FUNCTION_BLOCK EventWrapper_JACK2 (* Composite Function Block Type *)
  (* Standard: 61499-2 *)
  (* Version 0.0, 4/9/2019, erik, nxtControl GmbH, template *)
  PACKAGE Main;
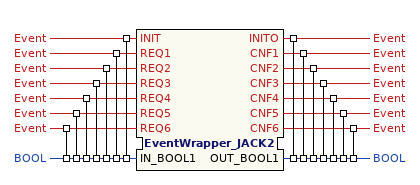
  EVENT_INPUT
    INIT WITH IN_BOOL1; (* Initialization Request *)
    REQ1 WITH IN_BOOL1; (* Normal Execution Request *)
    REQ2 WITH IN_BOOL1;
    REQ3 WITH IN_BOOL1;
    REQ4 WITH IN_BOOL1;
    REQ5 WITH IN_BOOL1;
    REQ6 WITH IN_BOOL1;
  END_EVENT
  EVENT_OUTPUT
    INITO WITH OUT_BOOL1; (* Initialization Confirm *)
    CNF1 WITH OUT_BOOL1; (* Execution Confirmation *)
    CNF2 WITH OUT_BOOL1;
    CNF3 WITH OUT_BOOL1;
    CNF4 WITH OUT_BOOL1;
    CNF5 WITH OUT_BOOL1;
    CNF6 WITH OUT_BOOL1;
  END_EVENT
  VAR_INPUT
    IN_BOOL1 : BOOL;
  END_VAR
  VAR_OUTPUT
    OUT_BOOL1 : BOOL;
  END_VAR
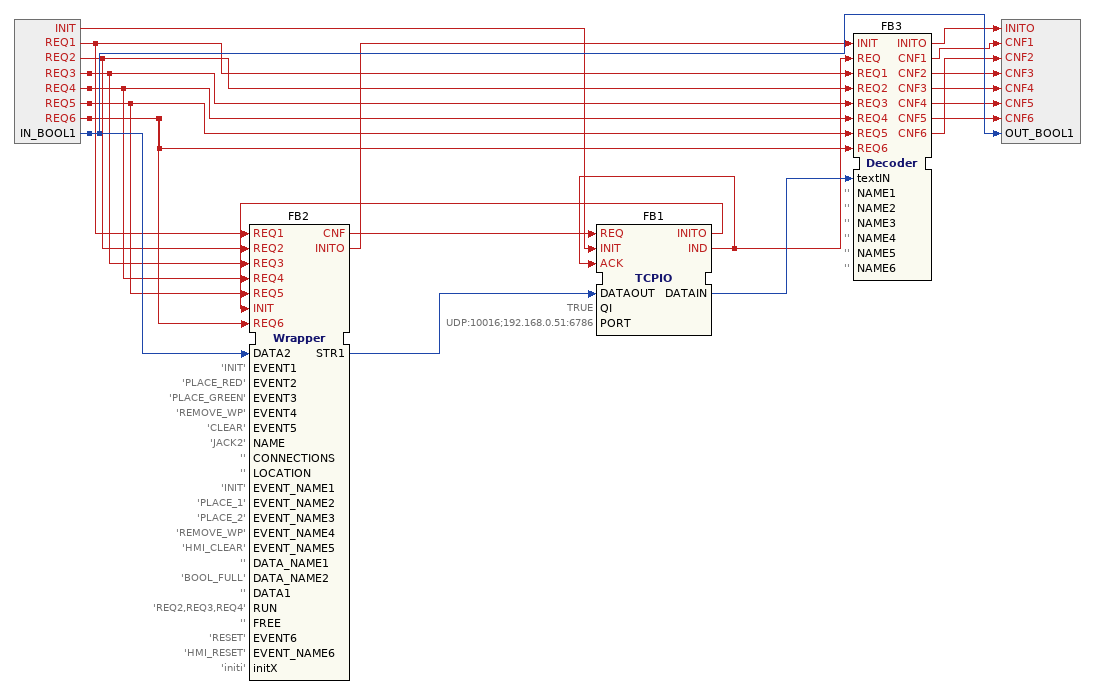
  FBS
    FB1 : TCPIO(QI := TRUE, PORT := UDP:10016;192.168.0.51:6786);
    FB2 : Wrapper(EVENT1 := 'INIT', EVENT2 := 'PLACE_RED', EVENT3 := 'PLACE_GREEN', EVENT4 := 'REMOVE_WP', EVENT5 := 'CLEAR', NAME := 'JACK2', CONNECTIONS := '', LOCATION := '', EVENT_NAME1 := 'INIT', EVENT_NAME2 := 'PLACE_1', EVENT_NAME3 := 'PLACE_2', EVENT_NAME4 := 'REMOVE_WP', EVENT_NAME5 := 'HMI_CLEAR', DATA_NAME1 := '', DATA_NAME2 := 'BOOL_FULL', DATA1 := '', RUN := 'REQ2,REQ3,REQ4', FREE := '', EVENT6 := 'RESET', EVENT_NAME6 := 'HMI_RESET', initX := 'initi');
    FB3 : Decoder(NAME1 := '', NAME2 := '', NAME3 := '', NAME4 := '', NAME5 := '', NAME6 := '');
  END_FBS
  EVENT_CONNECTIONS
    REQ1 TO FB2.REQ1;
    REQ2 TO FB2.REQ2;
    REQ3 TO FB2.REQ3;
    FB2.CNF TO FB1.REQ;
    REQ4 TO FB2.REQ4;
    REQ5 TO FB2.REQ5;
    INIT TO FB1.INIT;
    FB1.INITO TO FB2.INIT;
    FB1.IND TO FB1.ACK;
    REQ6 TO FB2.REQ6;
    FB1.IND TO FB3.REQ;
    FB3.INITO TO INITO;
    FB3.CNF3 TO CNF3;
    FB3.CNF2 TO CNF2;
    FB3.CNF1 TO CNF1;
    FB3.CNF4 TO CNF4;
    FB3.CNF5 TO CNF5;
    FB3.CNF6 TO CNF6;
    REQ1 TO FB3.REQ1;
    REQ2 TO FB3.REQ2;
    REQ3 TO FB3.REQ3;
    REQ4 TO FB3.REQ4;
    REQ5 TO FB3.REQ5;
    REQ6 TO FB3.REQ6;
    FB2.INITO TO FB3.INIT;
  END_CONNECTIONS
  DATA_CONNECTIONS
    FB2.STR1 TO FB1.DATAOUT;
    FB1.DATAIN TO FB3.textIN;
    IN_BOOL1 TO OUT_BOOL1;
    IN_BOOL1 TO FB2.DATA2;
  END_CONNECTIONS
END_FUNCTION_BLOCK
